// TIA Portal V20 export
DATA_BLOCK "DB_LogMsg"   // DB39
// stored: MemoryReserve 100, Namespace ProductionLine
   VAR
      Write_Position : Int;
      abyLogMsg_Buffer : Array[0..8191] of Byte;
      LogMsg_1 : Struct
         Para_BYTE_02 : "ProductionLine.Log_Data_Byte_Decimal";
      END_STRUCT;
      LogMsg_2 : Struct
         Para_BYTE_02 : "ProductionLine.Log_Data_Byte_Decimal";
      END_STRUCT;
      LogMsg_3 : Struct
         Para_BYTE_02 : "ProductionLine.Log_Data_Byte_Decimal";
      END_STRUCT;
      LogMsg_4 : Struct
         Para_STRING_01 : "ProductionLine.Log_Data_String20";
         Para_BYTE_02 : "ProductionLine.Log_Data_Byte_Decimal";
         Para_STRING_05 : "ProductionLine.Log_Data_String20";
      END_STRUCT;
      LogMsg_5 : Struct
         Para_STRING_01 : "ProductionLine.Log_Data_String20";
         Para_BYTE_02 : "ProductionLine.Log_Data_Byte_Decimal";
         Para_STRING_03 : "ProductionLine.Log_Data_String20";
         Para_STRING_05 : "ProductionLine.Log_Data_String20";
      END_STRUCT;
      LogMsg_6 : Struct
         Para_STRING_01 : "ProductionLine.Log_Data_String20";
         Para_BYTE_02 : "ProductionLine.Log_Data_Byte_Decimal";
      END_STRUCT;
      LogMsg_7 : Struct
         Para_STRING_01 : "ProductionLine.Log_Data_String20";
         Para_BYTE_02 : "ProductionLine.Log_Data_Byte_Decimal";
         Para_STRING_03 : "ProductionLine.Log_Data_String20";
         Para_STRING_04 : "ProductionLine.Log_Data_String20";
      END_STRUCT;
      LogMsg_8 : Struct
         Para_STRING_01 : "ProductionLine.Log_Data_String20";
         Para_BYTE_02 : "ProductionLine.Log_Data_Byte_Decimal";
      END_STRUCT;
      LogMsg_9 : Struct
         Para_STRING_01 : "ProductionLine.Log_Data_String20";
         Para_BYTE_02 : "ProductionLine.Log_Data_Byte_Decimal";
         Para_STRING_03 : "ProductionLine.Log_Data_String20";
         Para_STRING_04 : "ProductionLine.Log_Data_String20";
         Para_STRING_05 : "ProductionLine.Log_Data_String20";
      END_STRUCT;
      LogMsg_10 : Struct
         Para_STRING_01 : "ProductionLine.Log_Data_String20";
         Para_BYTE_02 : "ProductionLine.Log_Data_Byte_Decimal";
         Para_STRING_03 : "ProductionLine.Log_Data_String20";
         Para_STRING_04 : "ProductionLine.Log_Data_String20";
         Para_CHAR_05 : "ProductionLine.Log_Data_Char";
      END_STRUCT;
   END_VAR
BEGIN
END_DATA_BLOCK
